// TwinCAT 3 PLC project Main
// ProgramVersion: 3.1.4024.0
// libraries:
//   mobject-core, * (mobject)
//   Tc2_Standard, * (Beckhoff Automation GmbH)
//   Tc2_System, * (Beckhoff Automation GmbH)
//   Tc2_Utilities, * (Beckhoff Automation GmbH)
//   Tc3_Module, * (Beckhoff Automation GmbH)
//   Tc3_Vision, * (Beckhoff Automation GmbH)
//   TcUnit, * (www.tcunit.org)
// project tree:
//   / PlcTask.TcTTO
//   POUs/Library/Animation/ I_Animation.TcIO, SpriteSheetAnimationFrames.TcPOU
//   POUs/Library/EL2574/DUT/ EL2574_Command.TcDUT
//   POUs/Library/EL2574/ EL2574_ExtendedMode.TcPOU, EL2574_CommandMode.TcPOU, I_EL2574_CommandMode.TcIO
//   POUs/Library/Functions/ HtmlColorCodeToRGBA.TcPOU
//   POUs/Library/Scene/ Scene.TcPOU
//   POUs/Library/ImageSerializer/Base/ ImageSerializer.TcPOU
//   POUs/Library/ImageSerializer/Interfaces/ I_ImageSerializer.TcIO
//   POUs/Library/ImageSerializer/Matrix/ MatrixImageSerializer.TcPOU
//   POUs/Library/ImageSerializer/Null/ NullImageSerializer.TcPOU
//   POUs/Library/PixelReader/ I_PixelReader.TcIO, EL2574PixelReader.TcPOU
//   POUs/ MAIN.TcPOU
//   Tests/ EL2574PixelReader_TestSuite.TcPOU, UnitTests.TcPOU
// real-time tasks:
//   TASK PlcTask: cycle T#700us, priority 20, ADS port 350
// I/O:
//   DEVICE Device 3 (EtherCAT), AmsNetId 172.18.232.102.4.1
//     Term 1 (EK1100) [EK1100 EtherCAT Coupler (2A E-Bus)]
//       Term 2 (EL2004) [EL2004 4Ch. Dig. Output 24V, 0.5A]
//       Term 3 (EL1014) [EL1014 4Ch. Dig. Input 24V, 10µs]
//       Term 4 (EL2574) [EL2574 4 Ch. Pixel LED Controller]
//         modules: SlotGroup 1 (Slot 1, 2) (1xASYNC), SlotGroup 1 (Slot 1, 2) (1xASYNC), SlotGroup 2 (Slot 3, 4) (1xASYNC), SlotGroup 2 (Slot 3, 4) (1xASYNC)
//       Term 5 (EL9011) [EL9011 End Terminal]
// variable links:
//   Main Instance <-> Device 3 (EtherCAT)/Term 1 (EK1100)/Term 3 (EL1014)
//     PlcTask Inputs/MAIN.switch <-> Channel 1/Input
//   Main Instance <-> Device 3 (EtherCAT)/Term 1 (EK1100)/Term 4 (EL2574)
//     PlcTask Inputs/MAIN.el2574_ch1.pdo.MDP5001_260_Input/MDP5001_260_Status <-> SlotGroup 1 (Slot 1, 2) (1xASYNC)/Status Channel 1/Status
//     PlcTask Inputs/MAIN.el2574_ch3.pdo.MDP5001_260_Input/MDP5001_260_Status <-> SlotGroup 2 (Slot 3, 4) (1xASYNC)/Status Channel 1/Status
//     PlcTask Outputs/MAIN.el2574_ch1.pdo.MDP5001_260_Output/MDP5001_260_Extended_Control <-> SlotGroup 1 (Slot 1, 2) (1xASYNC)/Extended Channel 1/Extended Control
//     PlcTask Outputs/MAIN.el2574_ch3.pdo.MDP5001_260_Output/MDP5001_260_Control <-> SlotGroup 2 (Slot 3, 4) (1xASYNC)/Control Channel 1/Control

CONFIGURATION Main
    RESOURCE PLC ON TwinCAT3
        TASK PlcTask(INTERVAL := T#700us, PRIORITY := 20);
        PROGRAM MAIN WITH PlcTask : MAIN;
    END_RESOURCE
END_CONFIGURATION

// ---- POUs/Library/EL2574/DUT/EL2574_Command.TcDUT
TYPE EL2574_Command :
STRUCT
	Send : BOOL;
	Update : BOOL;
	Command : USINT;
	Index : UINT;
	Length : UINT;
	Parameter : UINT;
	ColorRed : USINT;
	ColorGreen : USINT;
	ColorBlue : USINT;
	ColorWhite : USINT;
END_STRUCT
END_TYPE

// ---- POUs/Library/Animation/I_Animation.TcIO
INTERFACE I_Animation

PROPERTY PUBLIC CurrentFrameImage : ITcVnImage
GET
END_GET
END_PROPERTY

PROPERTY PUBLIC CurrentFrameIndex : UDINT
GET
END_GET
END_PROPERTY

PROPERTY PUBLIC IsAtLastFrame : BOOL
GET
END_GET
END_PROPERTY

METHOD PUBLIC MoveToStart
VAR_INPUT
END_VAR
END_METHOD

PROPERTY PUBLIC TotalFrameCount : UDINT
GET
END_GET
END_PROPERTY

METHOD PUBLIC TryMoveNext : BOOL
VAR_INPUT
END_VAR
END_METHOD

METHOD PUBLIC TryMovePrevious : BOOL
VAR_INPUT
END_VAR
END_METHOD

END_INTERFACE

// ---- POUs/Library/EL2574/I_EL2574_CommandMode.TcIO
INTERFACE I_EL2574_CommandMode

METHOD PUBLIC ClearAll : I_EL2574_CommandMode
VAR_INPUT
END_VAR
END_METHOD

METHOD PUBLIC ColorGradient2Point : I_EL2574_CommandMode
VAR_INPUT
	StartPosition : UINT;
	NumberOfPixels : UINT;
	Color1 : STRING(9);
	Color2 : STRING(9);
END_VAR
END_METHOD

METHOD PUBLIC ColorGradient3Point : I_EL2574_CommandMode
VAR_INPUT
	StartPosition : UINT;
	NumberOfPixels : UINT;
	Color1 : STRING(9);
	Color2 : STRING(9);
	Color3 : STRING(9);
END_VAR
END_METHOD

METHOD PUBLIC ColorGradient4Point : I_EL2574_CommandMode
VAR_INPUT
	StartPosition : UINT;
	NumberOfPixels : UINT;
	Color1 : STRING(9);
	Color2 : STRING(9);
	Color3 : STRING(9);
	Color4 : STRING(9);
END_VAR
END_METHOD

METHOD PUBLIC CopyPixels : I_EL2574_CommandMode
VAR_INPUT
	StartPosition : UINT;
	NumberOfPixels : UINT;
	TargetPosition : UINT;
END_VAR
END_METHOD

METHOD PUBLIC FillColor : I_EL2574_CommandMode
VAR_INPUT
	StartPosition : UINT;
	NumberOfPixels : UINT;
	Red : USINT;
	Green : USINT;
	Blue : USINT;
	White : USINT;
END_VAR
END_METHOD

METHOD PUBLIC Invert : I_EL2574_CommandMode
VAR_INPUT
	StartPosition : UINT;
	NumberOfPixels : UINT;
END_VAR
END_METHOD

METHOD PUBLIC MovePixels : I_EL2574_CommandMode
VAR_INPUT
	StartPosition : UINT;
	NumberOfPixels : UINT;
	TargetPosition : UINT;
END_VAR
END_METHOD

METHOD PUBLIC RotateLeft : I_EL2574_CommandMode
VAR_INPUT
	StartPosition : UINT;
	NumberOfPixels : UINT;
	Shift : UINT;
END_VAR
END_METHOD

METHOD PUBLIC RotateRight : I_EL2574_CommandMode
VAR_INPUT
	StartPosition : UINT;
	NumberOfPixels : UINT;
	Shift : UINT;
END_VAR
END_METHOD

METHOD PUBLIC Send : I_EL2574_CommandMode
VAR_INPUT
END_VAR
END_METHOD

METHOD PUBLIC SendAndUpdate : I_EL2574_CommandMode
VAR_INPUT
END_VAR
END_METHOD

METHOD PUBLIC Update : I_EL2574_CommandMode
VAR_INPUT
END_VAR
END_METHOD

END_INTERFACE

// ---- POUs/Library/ImageSerializer/Interfaces/I_ImageSerializer.TcIO
INTERFACE I_ImageSerializer

METHOD PUBLIC ConnectTo
VAR_INPUT
	ImageSerializer : I_ImageSerializer;
END_VAR
END_METHOD

METHOD PUBLIC GetTotalSerializablePixelCount : UDINT
VAR_INPUT
END_VAR
END_METHOD

PROPERTY PUBLIC PixelCount : UDINT
GET
END_GET
END_PROPERTY

METHOD PUBLIC TryGetPixel : BOOL
VAR_INPUT
	PixelIndex : UDINT;
	Reader : I_PixelReader;
END_VAR
END_METHOD

METHOD PUBLIC UpdateImage
VAR_INPUT
	Source : ITcVnImage;
END_VAR
END_METHOD

END_INTERFACE

// ---- POUs/Library/PixelReader/I_PixelReader.TcIO
INTERFACE I_PixelReader

PROPERTY PUBLIC Value : Reference to TcVnVector4_LREAL
GET
END_GET
END_PROPERTY

END_INTERFACE

// ---- POUs/MAIN.TcPOU
PROGRAM MAIN
VAR
	// demo triggers
	startAnimation : BOOL := TRUE;
	clear : BOOL := FALSE;
	mode : (RANDOM, NAUGHTY, NICE, SPECIAL) := RANDOM; // defaults each time to random
	
	// animations
	fireAnimation : SpriteSheetAnimationFrames(
		SpriteSheetFilePath := 'C:\temp\FireplaceAndFire_2_3_6.png',
		SpriteWidth := 32,
		SpriteHeight := 32,
		TotalSprites := 6,
		Columns := 2,
		Rows := 3
	);
	
	idleAnimation : SpriteSheetAnimationFrames(
		SpriteSheetFilePath := 'C:\temp\NaughtyOrNiceOutline_5_6_29.png',
		SpriteWidth := 32,
		SpriteHeight := 32,
		TotalSprites := 29,
		Columns := 5,
		Rows := 6
	);
	
	checkingList : SpriteSheetAnimationFrames(
		SpriteSheetFilePath := 'C:\temp\CheckingElfTree_4_4_16.png',
		SpriteWidth := 32,
		SpriteHeight := 32,
		TotalSprites := 16,
		Columns := 4,
		Rows := 4
	);
	
	anyCoverAnimation : SpriteSheetAnimationFrames(
		SpriteSheetFilePath := 'C:\temp\AnyCover_4_4_16.png',
		SpriteWidth := 32,
		SpriteHeight := 32,
		TotalSprites := 16,
		Columns := 4,
		Rows := 4
	);
	
	grinchAnimation : SpriteSheetAnimationFrames(
		SpriteSheetFilePath := 'C:\temp\Grinch_4_4_15.png',
		SpriteWidth := 32,
		SpriteHeight := 32,
		TotalSprites := 15,
		Columns := 4,
		Rows := 4
	);
	
	nicePresentAnimation : SpriteSheetAnimationFrames(
		SpriteSheetFilePath := 'C:\temp\NicePresent_4_5_19.png',
		SpriteWidth := 32,
		SpriteHeight := 32,
		TotalSprites := 19,
		Columns := 4,
		Rows := 5
	);
	
	specialAnimation : SpriteSheetAnimationFrames(
		SpriteSheetFilePath := 'C:\temp\sp_3_4_12.png',
		SpriteWidth := 32,
		SpriteHeight := 32,
		TotalSprites := 12,
		Columns := 3,
		Rows := 4
	);

	// matrix panels
	matrix1 : MatrixImageSerializer(Height := 16, Width := 16, X := 16, Y := 16, FlipX := FALSE, FlipY := TRUE, Rotate := TRUE);
	matrix2 : MatrixImageSerializer(Height := 16, Width := 16, X := 16, Y := 0, FlipX := FALSE, FlipY := TRUE, Rotate := TRUE); 
	matrix3 : MatrixImageSerializer(Height := 16, Width := 16, X := 0, Y := 0, FlipX := FALSE, FlipY := TRUE, Rotate := TRUE); 
	matrix4 : MatrixImageSerializer(Height := 16, Width := 16, X := 0, Y := 16, FlipX := FALSE, FlipY := TRUE, Rotate := TRUE); 
	
	// helpers
	scene : Scene;
	
	// hardware
	switch AT %I* : BOOL;
	el2574_ch1 : EL2574_ExtendedMode(TotalPixels := 1024); // you need to pass in the total number of pixels connected to the EK2574
	el2574_ch3 : EL2574_CommandMode(TotalPixels := 1024);
	
	// program variables
	initialized : BOOL;
	
	animationState : (
		IDLE_FWD, 
		IDLE_FWD_WAIT, 
		IDLE_BACKWARD, 
		IDLE_BACKWARD_WAIT, 
		CHECK_LIST, 
		COVER, 
		REVEAL_DECIDE, 
		REVEAL, 
		ACTUAL, 
		END_DELAY, 
		RESET
	) := RESET;
	
	actualAnimation : I_Animation;
	decision : USINT;
	
	ledState : (OFF, 
		OFF_WAIT, 
		IDLE_START, 
		IDLE_SEND_NEXT, 
		IDLE_WAIT, 
		CHECKING_START, 
		CHECKING_SEND_NEXT, 
		CHECKING_WAIT, 
		COVER_START,
		COVER_SEND_NEXT, 
		COVER_WAIT,
		REVEAL_NAUGHTY_START, 
		REVEAL_NAUGHTY_SEND_NEXT, 
		REVEAL_NAUGHTY_WAIT,
		REVEAL_NICE_START, 
		REVEAL_NICE_SEND_NEXT, 
		REVEAL_NICE_WAIT,
		REVEAL_SPECIAL_START, 
		REVEAL_SPECIAL_SEND_NEXT, 
		REVEAL_SPECIAL_WAIT
	) := OFF;
	
	animationRTrigger : R_TRIG;
	switchRTrigger : R_TRIG;
	triggerLedOff : R_TRIG;
	triggerLedIdle : R_TRIG;
	triggerLedChecking : R_TRIG;
	triggerLedCover : R_TRIG;
	triggerLedReveal : R_TRIG;
	
	// randomizer
	randomizer : USINT := 1; // very basic randomizer
	
	// counters 
	checklistCounter : INT; // this is just a simple setup to slow the animation down
	
	// timers
	idleForwardTimer : TON := (PT:=T#1S);
	idleBackwardTimer : TON := (PT:=T#2S);
	revealDecideTimer : TON := (PT:=T#1S);
	endDelayTimer : TON := (PT:=T#3S);
	fastLedTickerTimer : TON := (PT:=T#50MS);
	slowLedTickerTimer : TON := (PT:=T#200MS);
	
	// colors - variables so I can set them for testing. 	
	IDLE_COLOR_1 : STRING(9) := '04eeff';
	IDLE_COLOR_2 : STRING(9) := 'a206b1';
	IDLE_COLOR_3 : STRING(9) := '04eeff';
	
	CHECKING_COLOR_1 : STRING(9) := '0314f8';
	CHECKING_COLOR_2 : STRING(9) := '50aaa3';
	CHECKING_COLOR_3 : STRING(9) := '0314f8';

	COVER_COLOR_1 : STRING(9) := '09860f';
	COVER_COLOR_2 : STRING(9) := 'FF0000';
	COVER_COLOR_3 : STRING(9) := '09860f';
	
	REVEAL_NAUGHTY_COLOR_1 : STRING(9) := '09860f';
	REVEAL_NAUGHTY_COLOR_2 : STRING(9) := '000000';
	REVEAL_NAUGHTY_COLOR_3 : STRING(9) := '09860f';
	
	REVEAL_NICE_COLOR_1 : STRING(9) := 'FF0000';
	REVEAL_NICE_COLOR_2 : STRING(9) := '222222';
	REVEAL_NICE_COLOR_3 : STRING(9) := 'FF0000';
	
	REVEAL_SPECIAL_COLOR_1 : STRING(9) := 'f3ef16';
	REVEAL_SPECIAL_COLOR_2 : STRING(9) := 'FF0000';
	REVEAL_SPECIAL_COLOR_3 : STRING(9) := 'f3ef16';

END_VAR
VAR CONSTANT
	LED_STRIP_START : UINT := 120;
	LED_STRIP_LENGTH : UINT := 178;
END_VAR

(*

  _____ __  __ _____   ____  _____ _______       _   _ _______ _ 
 |_   _|  \/  |  __ \ / __ \|  __ \__   __|/\   | \ | |__   __| |
   | | | \  / | |__) | |  | | |__) | | |  /  \  |  \| |  | |  | |
   | | | |\/| |  ___/| |  | |  _  /  | | / /\ \ | . ` |  | |  | |
  _| |_| |  | | |    | |__| | | \ \  | |/ ____ \| |\  |  | |  |_|
 |_____|_|  |_|_|     \____/|_|  \_\ |_/_/    \_\_| \_|  |_|  (_)
 
Competition Clause: 

During the Beckhoff Christmas coding competition involving the EL2574 
LED controller terminal, if any Beckhoff subsidiaries use, borrow from, or are inspired
by this code for their own competition entry, they must acknowledge the inspiration by 
including the hashtag #codingbytes in any LinkedIn posts related to their competition entry. 
This requirement is in effect until the conclusion OF the competition on 25th December 2024.

*)

IF NOT initialized THEN
	// First setup the wiring of the units.  This must be in the order they are physically connected.
	matrix1.ConnectTo(matrix2);
	matrix2.ConnectTo(matrix3);
	matrix3.ConnectTo(matrix4);
	// that's initializing done!
	initialized := TRUE;
END_IF

// we wait here until the animation source image is loaded.
// i.e. we return, which prevents the program from progressing past this line.
IF NOT specialAnimation.TryLoad() OR NOT fireAnimation.TryLoad() OR NOT idleAnimation.TryLoad() OR NOT checkingList.TryLoad() OR NOT anyCoverAnimation.TryLoad() OR NOT grinchAnimation.TryLoad() OR NOT nicePresentAnimation.TryLoad() THEN
    RETURN;
END_IF

// basic clear trigger.  Set clear TRUE to clear the display
IF clear AND_THEN el2574_ch1.TrySendClearAll() THEN
	clear := FALSE;
END_IF

// if the startAnimation flag is triggered then force the state machine to RESET
animationRTrigger(Clk:=startAnimation);
IF animationRTrigger.Q THEN
	animationState := RESET;
END_IF

// if the "check" switch is pulled then move to CHECK_LIST if the program is running in idle
switchRTrigger(clk:=switch);
IF startAnimation AND switchRTrigger.Q AND (animationState = IDLE_FWD OR animationState = IDLE_FWD_WAIT OR animationState = IDLE_BACKWARD OR animationState = IDLE_BACKWARD_WAIT) THEN
	animationState := CHECK_LIST;
	decision := randomizer;
END_IF 

// animation state machine.
// this controls all of the image, animation and timinigs. 
IF startAnimation  AND NOT el2574_ch1.IsBusy THEN 
	
	CASE animationState OF
	
		IDLE_FWD :
			
			scene.Initalize(fireAnimation.CurrentFrameImage);
			scene.AddLayer(idleAnimation.CurrentFrameImage);
			
			IF NOT fireAnimation.TryMoveNext() THEN
				fireAnimation.MoveToStart();
			END_IF
			
			IF NOT idleAnimation.TryMoveNext() THEN
				animationState := IDLE_FWD_WAIT;
			END_IF
			
		IDLE_FWD_WAIT : 
		
			scene.Initalize(fireAnimation.CurrentFrameImage);
			scene.AddLayer(idleAnimation.CurrentFrameImage);
			
			IF NOT fireAnimation.TryMoveNext() THEN
				fireAnimation.MoveToStart();
			END_IF
		
			IF idleForwardTimer.Q THEN
				animationState := IDLE_BACKWARD;
			END_IF

		IDLE_BACKWARD :  
		
			scene.Initalize(fireAnimation.CurrentFrameImage);
			scene.AddLayer(idleAnimation.CurrentFrameImage);
			
			IF NOT fireAnimation.TryMoveNext() THEN
				fireAnimation.MoveToStart();
			END_IF
			
			IF NOT idleAnimation.TryMovePrevious() THEN
				animationState := IDLE_BACKWARD_WAIT;
			END_IF	

		IDLE_BACKWARD_WAIT : //	
		
			scene.Initalize(fireAnimation.CurrentFrameImage);
			scene.AddLayer(idleAnimation.CurrentFrameImage);
			
			IF NOT fireAnimation.TryMoveNext() THEN
				fireAnimation.MoveToStart();
			END_IF
		
			IF idleBackwardTimer.Q THEN
				animationState := IDLE_FWD;
			END_IF
			
		CHECK_LIST : 
		
			scene.Initalize(checkingList.CurrentFrameImage);
			
			IF checklistCounter > 2 AND_THEN NOT checkingList.TryMoveNext() THEN
				animationState := COVER;
			END_IF
			
			IF checklistCounter > 2 THEN
				checklistCounter := 0;
			ELSE 
				checklistCounter := checklistCounter + 1;
			END_IF
		
		COVER : //
		
			scene.Initalize(checkingList.CurrentFrameImage);
			scene.AddLayer(anyCoverAnimation.CurrentFrameImage);
			
			IF not anyCoverAnimation.TryMoveNext() THEN
				animationState := REVEAL_DECIDE;
			END_IF
			
		REVEAL_DECIDE : //
		
			IF revealDecideTimer.Q THEN
				
				// change mode to one of the two randoms.
				IF mode = RANDOM THEN
					IF decision > 5 THEN
						mode := NAUGHTY;
					ELSE
						mode := NICE;
					END_IF
				END_IF
				
				IF mode = NAUGHTY THEN
					actualAnimation := grinchAnimation;
				ELSIF mode = NICE THEN
					actualAnimation := nicePresentAnimation;
				ELSIF mode = SPECIAL THEN
					actualAnimation := specialAnimation;
				END_IF

				animationState := REVEAL;

			END_IF
		
		REVEAL : //
		
			scene.Initalize(actualAnimation.CurrentFrameImage);
			scene.AddLayer(anyCoverAnimation.CurrentFrameImage);
			
			IF NOT anyCoverAnimation.TryMovePrevious() THEN
				animationState := ACTUAL;
			END_IF
		
		ACTUAL : // 
		
			scene.Initalize(actualAnimation.CurrentFrameImage);
			
			IF NOT actualAnimation.TryMoveNext() THEN
				animationState := END_DELAY;
			END_IF
			
		END_DELAY : //
		
			IF endDelayTimer.Q THEN
				animationState := RESET;
			END_IF
			
		RESET : //
		
			idleAnimation.MoveToStart();
			checkingList.MoveToStart();
			anyCoverAnimation.MoveToStart();
			grinchAnimation.MoveToStart();
			nicePresentAnimation.MoveToStart();
			animationState := IDLE_FWD;
			mode := RANDOM;
	
	END_CASE
	
	matrix1.UpdateImage(scene.Image);
	el2574_ch1.TrySendPixelsFromSerializer(matrix1);
	
END_IF

// naughty, nice randomizer
randomizer := randomizer + 1;
IF randomizer > 10 THEN 
	randomizer := 1;
END_IF

// timers
idleForwardTimer(IN:=animationState=IDLE_FWD_WAIT);
idleBackwardTimer(IN:=animationState=IDLE_BACKWARD_WAIT);
revealDecideTimer(IN:=animationState=REVEAL_DECIDE);
endDelayTimer(IN:=animationState=END_DELAY);
fastLedTickerTimer(IN:=NOT fastLedTickerTimer.Q);
slowLedTickerTimer(IN:=NOT slowLedTickerTimer.Q);

// led state triggers
triggerLedOff(CLK := animationState=RESET);
IF triggerLedOff.Q THEN
	ledState := OFF;
END_IF

triggerLedIdle(CLK := animationState=IDLE_FWD);
IF triggerLedIdle.Q THEN
	ledState := IDLE_START;
END_IF

triggerLedChecking(CLK := animationState=CHECK_LIST);
IF triggerLedChecking.Q THEN
	ledState := CHECKING_START;
END_IF

triggerLedCover(CLK := animationState=COVER);
IF triggerLedCover.Q THEN
	ledState := COVER_START;
END_IF

triggerLedReveal(CLK := animationState=ACTUAL);
IF triggerLedReveal.Q THEN
	IF mode = NAUGHTY THEN
		ledState := REVEAL_NAUGHTY_START;
	ELSIF mode = NICE THEN
		ledState := REVEAL_NICE_START;
	ELSIF mode = SPECIAL THEN
		ledState := REVEAL_SPECIAL_START;
	END_IF
END_IF


// led state machine
CASE ledState OF
	
	OFF : //
	
		el2574_ch3.ClearAll();
		el2574_ch3.SendAndUpdate();
		ledState := OFF_WAIT;
	
	OFF_WAIT : // 
	
	IDLE_START : //
	
		el2574_ch3.ClearAll();
		el2574_ch3.ColorGradient3Point(LED_STRIP_START, 180, IDLE_COLOR_1, IDLE_COLOR_2, IDLE_COLOR_3);
		el2574_ch3.SendAndUpdate();
		ledState := IDLE_SEND_NEXT;
	
	IDLE_SEND_NEXT : //
	
		el2574_ch3.RotateRight(LED_STRIP_START, 180, 1); 
		el2574_ch3.SendAndUpdate();
		ledState := IDLE_WAIT;
		
	IDLE_WAIT : //
	
		IF NOT el2574_ch3.IsBusy AND fastLedTickerTimer.Q THEN
			ledState := IDLE_SEND_NEXT;
		END_IF
		
	CHECKING_START : //
	
		el2574_ch3.ClearAll();
		el2574_ch3.ColorGradient3Point(LED_STRIP_START, 180, CHECKING_COLOR_1, CHECKING_COLOR_2, CHECKING_COLOR_3);
		ledState := CHECKING_SEND_NEXT;
	
	CHECKING_SEND_NEXT : //
	
		el2574_ch3.RotateRight(LED_STRIP_START, 180, 1); 
		el2574_ch3.SendAndUpdate();
		ledState := CHECKING_WAIT;
	
	CHECKING_WAIT : //
	
		IF NOT el2574_ch3.IsBusy THEN
			ledState := CHECKING_SEND_NEXT;
		END_IF
		
	COVER_START : //
	
		el2574_ch3.ClearAll();
		el2574_ch3.ColorGradient3Point(LED_STRIP_START, 180, COVER_COLOR_1, COVER_COLOR_2, COVER_COLOR_3);
		ledState := COVER_SEND_NEXT;
	
	COVER_SEND_NEXT : //
	
		el2574_ch3.RotateRight(LED_STRIP_START, 180, 1); 
		el2574_ch3.SendAndUpdate();
		ledState := COVER_WAIT;
	
	COVER_WAIT : //
	
		IF NOT el2574_ch3.IsBusy THEN
			ledState := COVER_SEND_NEXT;
		END_IF
		
	REVEAL_NAUGHTY_START : //
	
		el2574_ch3.ClearAll();
		el2574_ch3.ColorGradient3Point(LED_STRIP_START, 180, REVEAL_NAUGHTY_COLOR_1, REVEAL_NAUGHTY_COLOR_2, REVEAL_NAUGHTY_COLOR_3);
		ledState := REVEAL_NAUGHTY_SEND_NEXT;
	
	REVEAL_NAUGHTY_SEND_NEXT : //
	
		el2574_ch3.RotateRight(LED_STRIP_START, 180, 1); 
		el2574_ch3.SendAndUpdate();
		ledState := REVEAL_NAUGHTY_WAIT;
	
	REVEAL_NAUGHTY_WAIT : //
	
		IF NOT el2574_ch3.IsBusy THEN
			ledState := REVEAL_NAUGHTY_SEND_NEXT;
		END_IF
		
	REVEAL_NICE_START : //
	
		el2574_ch3.ClearAll();
		el2574_ch3.ColorGradient3Point(LED_STRIP_START, 180, REVEAL_NICE_COLOR_1, REVEAL_NICE_COLOR_2, REVEAL_NICE_COLOR_3);
		ledState := REVEAL_NICE_SEND_NEXT;
	
	REVEAL_NICE_SEND_NEXT : //
	
		el2574_ch3.RotateRight(LED_STRIP_START, 180, 1); 
		el2574_ch3.SendAndUpdate();
		ledState := REVEAL_NICE_WAIT;
	
	REVEAL_NICE_WAIT : //
	
		IF NOT el2574_ch3.IsBusy THEN
			ledState := REVEAL_NICE_SEND_NEXT;
		END_IF
		
	REVEAL_SPECIAL_START : //
	
		el2574_ch3.ClearAll();
		el2574_ch3.ColorGradient3Point(LED_STRIP_START, 180, REVEAL_SPECIAL_COLOR_1, REVEAL_SPECIAL_COLOR_2, REVEAL_SPECIAL_COLOR_3);
		ledState := REVEAL_SPECIAL_SEND_NEXT;
	
	REVEAL_SPECIAL_SEND_NEXT : //
	
		el2574_ch3.RotateRight(LED_STRIP_START, 180, 1); 
		el2574_ch3.SendAndUpdate();
		ledState := REVEAL_SPECIAL_WAIT;
	
	REVEAL_SPECIAL_WAIT : //
	
		IF NOT el2574_ch3.IsBusy THEN
			ledState := REVEAL_SPECIAL_SEND_NEXT;
		END_IF
		
END_CASE

// cyclic call the terminal so that it can do it's job.
el2574_ch1.CyclicCall();
el2574_ch3.CyclicCall();

// unit tests
UnitTests();

END_PROGRAM

// ---- POUs/Library/Animation/SpriteSheetAnimationFrames.TcPOU
FUNCTION_BLOCK SpriteSheetAnimationFrames implements I_Animation
VAR
	spriteSheetFilePath : T_MAXSTRING;
	spriteWidth : UDINT;
	spriteHeight : UDINT;
	totalSprites : UDINT;
	columns : UDINT;
	rows : UDINT;
	spriteSheetImage : ITcVnImage;
	readImage: FB_VN_ReadImage;
	
	// animation variables
	_currentFrameIndex : UDINT;
	_currentFrameImage : ITcVnImage;
END_VAR

PROPERTY PUBLIC CurrentFrameImage : ITcVnImage
GET
CurrentFrameImage := _currentFrameImage;
END_GET
END_PROPERTY

PROPERTY PUBLIC CurrentFrameIndex : UDINT
GET
CurrentFrameIndex := _currentFrameIndex;
END_GET
END_PROPERTY

METHOD FB_init : BOOL
VAR_INPUT
	bInitRetains : BOOL; // if TRUE, the retain variables are initialized (warm start / cold start)
	bInCopyCode : BOOL;  // if TRUE, the instance afterwards gets moved into the copy code (online change)
	SpriteSheetFilePath : T_MAXSTRING;
	SpriteWidth : UDINT;
	SpriteHeight : UDINT;
	TotalSprites : UDINT;
	Columns : UDINT;
	Rows : UDINT;
END_VAR
THIS^.spriteSheetFilePath := SpriteSheetFilePath;
THIS^.spriteWidth := SpriteWidth;
THIS^.spriteHeight := SpriteHeight;
THIS^.totalSprites := TotalSprites;
THIS^.columns := Columns;
THIS^.rows := Rows;
END_METHOD

PROPERTY PUBLIC IsAtLastFrame : BOOL
GET
IF TotalFrameCount = 0 THEN
	IsAtLastFrame := TRUE;
	RETURN;
END_IF

IsAtLastFrame := CurrentFrameIndex = TotalFrameCount - 1;
END_GET
END_PROPERTY

METHOD PUBLIC MoveToStart
VAR_INPUT
END_VAR
_currentFrameIndex := 0;
TryGetSprite(_currentFrameIndex, _currentFrameImage);
END_METHOD

PROPERTY PUBLIC TotalFrameCount : UDINT
GET
TotalFrameCount := totalSprites;
END_GET
END_PROPERTY

METHOD PRIVATE TryGetSprite : BOOL
VAR_INPUT
	Index : UDINT;
	Destination : REFERENCE TO ITcVnImage;
END_VAR
VAR
	spriteX : UDINT;
	spriteY : UDINT;
	spriteColumn : UDINT;
	spriteRow : UDINT;
	result : HRESULT;
END_VAR
IF Index > TotalFrameCount - 1 THEN
	RETURN;
END_IF

spriteColumn := Index MOD columns;
spriteRow := Index / columns;

spriteX := spriteColumn * spriteWidth;
spriteY := spriteRow * spriteHeight;

result := F_VN_CopyImage(spriteSheetImage, _currentFrameImage, s_OK);
result := F_VN_SetRoi(spriteX, spriteY, spriteWidth, spriteHeight, _currentFrameImage, result);

TryGetSprite := Succeeded(result);
END_METHOD

METHOD PUBLIC TryLoad : BOOL
VAR
	i : UDINT;
END_VAR
// if we already have an image loaded, then we can early jump out as we know everything is done. 
IF spriteSheetImage <> 0 THEN
	TryLoad := TRUE;
	RETURN;
END_IF

IF spriteSheetFilePath = '' OR  spriteWidth = 0 OR spriteHeight = 0 OR totalSprites = 0 OR columns = 0 OR rows = 0 THEN
	// this is our sanity check, we return out if anything is bad.
	// if we pass this point we know we can use the variables confidently.
	RETURN;
END_IF

// we keep polling the read until an image is read.  If it faults due to error then we just sit here and never return true.
readImage(sFilePath := spriteSheetFilePath, ipDestImage := spriteSheetImage, bRead := TRUE, nTimeout := T#500MS);
IF readImage.bBusy THEN 
	RETURN;
END_IF

IF readImage.bError THEN 
	RETURN;
END_IF 

// at this point we should have an image, so we will do one final check before moving on.  
IF spriteSheetImage = 0 THEN
	RETURN;
END_IF

// we have made it this far, which means we need to set the CurrentFrameImage to the first part of the image and report as done. 
MoveToStart();
TryLoad := TRUE;
END_METHOD

METHOD PUBLIC TryMoveNext : BOOL
VAR_INPUT
END_VAR
IF _currentFrameIndex = TotalFrameCount - 1 THEN
	RETURN;
END_IF

_currentFrameIndex := _currentFrameIndex + 1;
TryMoveNext := TryGetSprite(_currentFrameIndex, _currentFrameImage);
END_METHOD

METHOD PUBLIC TryMovePrevious : BOOL
VAR_INPUT
END_VAR
IF _currentFrameIndex = 0 THEN
	RETURN;
END_IF

_currentFrameIndex := _currentFrameIndex - 1;
TryMovePrevious := TryGetSprite(_currentFrameIndex, _currentFrameImage);
END_METHOD

END_FUNCTION_BLOCK

// ---- POUs/Library/ImageSerializer/Matrix/MatrixImageSerializer.TcPOU
FUNCTION_BLOCK MatrixImageSerializer EXTENDS ImageSerializer
VAR
	height : UDINT;
	width : UDINT;
	x : UDINT;
	y : UDINT;
	flipRequired : BOOL;
	flipAxis : ETcVnFlipAxis;
	rotateRequired : BOOL;
	rotateAngle : ETcVnRotationAngle;
	
	image : ITcVnImage;
	live : ITcVnDisplayableImage; // used in this demo to show the image for the matrix
	_pixelCount : UDINT;
END_VAR

METHOD FB_init : BOOL
VAR_INPUT
	bInitRetains : BOOL; // if TRUE, the retain variables are initialized (warm start / cold start)
	bInCopyCode : BOOL;  // if TRUE, the instance afterwards gets moved into the copy code (online change)
	Height : UDINT;
	Width : UDINT;
	X : UDINT;
	Y : UDINT;
	FlipX : BOOL;
	FlipY : BOOL;
	Rotate : BOOL;
END_VAR
THIS^.height := Height;
THIS^.width := Width;
THIS^.x := X;
THIS^.y := Y;

IF FlipX AND FlipY THEN
	flipAxis := ETcVnFlipAxis.TCVN_FA_XY;
	flipRequired := TRUE;
ELSIF FlipX THEN
	flipAxis := ETcVnFlipAxis.TCVN_FA_X;
	flipRequired := TRUE;
ELSIF FlipY THEN
	flipAxis := ETcVnFlipAxis.TCVN_FA_Y;
	flipRequired := TRUE;
END_IF

IF Rotate THEN
	rotateRequired := TRUE;
	rotateAngle := ETcVnRotationAngle.TCVN_RA_90_DEG;
END_IF

Initialize();
END_METHOD

METHOD PRIVATE Initialize
VAR_INPUT
END_VAR
_pixelCount := width * height;
END_METHOD

METHOD PROTECTED OnTryGetPixel : BOOL
VAR_INPUT
	PixelIndex : UDINT;
	Reader : I_PixelReader;
END_VAR
VAR
	xPosition : UDINT;
	yPosition : UDINT;
END_VAR
IF width = 0 OR height = 0 THEN
	RETURN;
END_IF

xPosition := PixelIndex MOD width;
yPosition := PixelIndex / width;

// If it's an odd row, reverse the direction
IF yPosition MOD 2 = 1 THEN 
    xPosition := (width - 1) - xPosition;
END_IF

OnTryGetPixel := succeeded(F_VN_GetPixel(image, Reader.Value, xPosition, yPosition, s_OK));
END_METHOD

METHOD PROTECTED OnUpdateImage
VAR_INPUT
	Source : ITcVnImage;
END_VAR
VAR
	result : HRESULT;
END_VAR
result := F_VN_CopyImage(Source, image, s_OK);
result := F_VN_SetRoi(x, y, width, height, image, result);

IF flipRequired THEN
	result := F_VN_FlipImage(image, image, flipAxis, result);	
END_IF

IF rotateRequired THEN
	result := F_VN_RotateImage(image, image, rotateAngle, result);	
END_IF

IF Succeeded(result) THEN
	F_VN_CopyIntoDisplayableImage(image, live, s_ok);
	RETURN;
END_IF

// there was an error, so best to clear the internal image as it's no longer valid.
// but only if there was an image there in fht first place.

IF image = 0 THEN
	RETURN;
END_IF

image.TcRelease();
image := 0;
END_METHOD

{attribute 'monitoring' := 'call'}
PROPERTY PUBLIC PixelCount : UDINT
GET
PixelCount := _pixelCount;
END_GET
END_PROPERTY

END_FUNCTION_BLOCK

// ---- POUs/Library/ImageSerializer/Base/ImageSerializer.TcPOU
FUNCTION_BLOCK ABSTRACT ImageSerializer IMPLEMENTS I_ImageSerializer
VAR
	// using the null object pattern so that you no longer need to check to see if next is <> 0
	nullImageSerializer : NullImageSerializer;
	next : I_ImageSerializer := nullImageSerializer;
END_VAR

METHOD PUBLIC ConnectTo
VAR_INPUT
	ImageSerializer : I_ImageSerializer;
END_VAR
IF ImageSerializer = 0  THEN
	next := nullImageSerializer;
END_IF

IF ImageSerializer = next THEN
	RETURN;
END_IF

next := ImageSerializer;
END_METHOD

METHOD PUBLIC GetTotalSerializablePixelCount : UDINT
VAR_INPUT
END_VAR
GetTotalSerializablePixelCount := PixelCount + NextSerializer.GetTotalSerializablePixelCount();
END_METHOD

PROPERTY PUBLIC NextSerializer : I_ImageSerializer
GET
NextSerializer := next;
END_GET
END_PROPERTY

METHOD PROTECTED ABSTRACT OnTryGetPixel : BOOL
VAR_INPUT
	PixelIndex : UDINT;
	Reader : I_PixelReader;
END_VAR
END_METHOD

METHOD PROTECTED ABSTRACT OnUpdateImage
VAR_INPUT
	Source : ITcVnImage;
END_VAR
END_METHOD

PROPERTY PUBLIC ABSTRACT PixelCount : UDINT
GET
END_GET
END_PROPERTY

METHOD PUBLIC TryGetPixel : BOOL
VAR_INPUT
	PixelIndex : UDINT;
	Reader : I_PixelReader;
END_VAR
VAR
	newPixelIndex : UDINT;
END_VAR
IF PixelIndex > PixelCount - 1 THEN
	newPixelIndex := PixelIndex - PixelCount;
	TryGetPixel := NextSerializer.TryGetPixel(newPixelIndex, Reader);
	RETURN;
END_IF

TryGetPixel := OnTryGetPixel(PixelIndex, Reader);
END_METHOD

METHOD PUBLIC UpdateImage
VAR_INPUT
	Source : ITcVnImage;
END_VAR
IF Source = 0 THEN
	RETURN;
END_IF

OnUpdateImage(Source);
NextSerializer.UpdateImage(Source);
END_METHOD

END_FUNCTION_BLOCK

// ---- POUs/Library/ImageSerializer/Null/NullImageSerializer.TcPOU
FUNCTION_BLOCK NullImageSerializer IMPLEMENTS I_ImageSerializer
VAR
END_VAR

METHOD PUBLIC ConnectTo
VAR_INPUT
	ImageSerializer : I_ImageSerializer;
END_VAR
END_METHOD

METHOD PUBLIC GetTotalSerializablePixelCount : UDINT
VAR_INPUT
END_VAR
GetTotalSerializablePixelCount := 0;
END_METHOD

PROPERTY PUBLIC PixelCount : UDINT
GET
PixelCount := 0;
END_GET
END_PROPERTY

METHOD PUBLIC TryGetPixel : BOOL
VAR_INPUT
	PixelIndex : UDINT;
	Reader : I_PixelReader;
END_VAR
TryGetPixel := FALSE;
END_METHOD

METHOD PUBLIC UpdateImage
VAR_INPUT
	Source : ITcVnImage;
END_VAR
END_METHOD

END_FUNCTION_BLOCK

// ---- POUs/Library/Scene/Scene.TcPOU
FUNCTION_BLOCK Scene
VAR
	sceneImage : ITcVnImage;
END_VAR

METHOD PUBLIC AddLayer
VAR_INPUT
	Source : ITcVnImage;
END_VAR
VAR
	sourceHeight, currentHeight : UDINT;
	sourceWidth, currentWidth : UDINT;
	x, y : UDINT;
	currentPixel : TcVnVector4_LREAL;
END_VAR
IF sceneImage = 0 THEN
	RETURN;
END_IF

IF Source = 0 THEN 
	RETURN;
END_IF

IF FAILED(Source.GetHeight(sourceHeight)) THEN
	RETURN;
END_IF;

IF FAILED(sceneImage.GetHeight(currentHeight)) THEN
	RETURN;
END_IF;

IF FAILED(Source.GetWidth(sourceWidth)) THEN
	RETURN;
END_IF;

IF FAILED(sceneImage.GetWidth(currentWidth)) THEN
	RETURN;
END_IF;

IF sourceHeight > currentHeight THEN
	RETURN;
END_IF

IF sourceWidth > currentWidth THEN
	RETURN;
END_IF

FOR y := 0 TO sourceHeight - 1 DO
	FOR x := 0 TO sourceWidth - 1 DO
		
		IF SUCCEEDED(F_VN_GetPixel(Source, currentPixel, x, y, s_OK)) THEN
			IF currentPixel[0] = 0 AND currentPixel[1] = 0 AND currentPixel[2] = 0 THEN
				CONTINUE;
			END_IF
			F_VN_SetPixel(sceneImage, currentPixel,x,y,s_OK);	
		END_IF
	
	END_FOR
END_FOR
END_METHOD

PROPERTY PUBLIC Image : ITcVnImage
GET
Image := sceneImage;
END_GET
END_PROPERTY

METHOD PUBLIC Initalize
VAR_INPUT
	Source : ITcVnImage;
END_VAR
F_VN_CopyImage(Source, sceneImage, s_OK);
END_METHOD

END_FUNCTION_BLOCK

// ---- POUs/Library/EL2574/EL2574_ExtendedMode.TcPOU
FUNCTION_BLOCK EL2574_ExtendedMode
VAR
	totalPixels : UDINT;
	pdo : MDP5001_260_80E6114C;
	sendBuffer : ARRAY [0..MAX_PIXELS - 1] OF UDINT;
	sendSegmentCount : USINT;
	currentSegment : USINT;
	state : (IDLE, INITIALIZING, SEND_SEGMENT, TRIGGER_FRAME_SEND, WAIT_FOR_FRAME_SEND_COMPLETE, ERROR);
END_VAR
VAR CONSTANT
	MAX_PIXELS : UDINT := 2048;
END_VAR

METHOD PRIVATE CreateSendBufferFromSerializer
VAR_INPUT
	ImageSerializer : I_ImageSerializer;
END_VAR
VAR
	currentPixel : UDINT := 0;
	pixelReader : EL2574PixelReader;
END_VAR
WHILE ImageSerializer.TryGetPixel(currentPixel, pixelReader) DO
	sendBuffer[currentPixel] := pixelReader.ReadAsUdint();
	currentPixel := currentPixel + 1;
END_WHILE
END_METHOD

METHOD PUBLIC CyclicCall
VAR_INPUT
END_VAR
VAR
	totalSegments : UDINT;
END_VAR
CASE state OF
	
	IDLE : RETURN;
	ERROR : RETURN;
	
	INITIALIZING :
	
		// initialize local variables
		currentSegment := 0;
		totalSegments := totalPixels / 8;
		sendSegmentCount := UDINT_TO_USINT(totalSegments);
	
		// reset the card to a known state
		pdo.MDP5001_260_Output.MDP5001_260_Extended_Control.Index := 0;
		pdo.MDP5001_260_Output.MDP5001_260_Extended_Control.Send := FALSE;
		pdo.MDP5001_260_Output.MDP5001_260_Extended_Control.Update := FALSE;
		pdo.MDP5001_260_Output.MDP5001_260_Extended_Control.Write := FALSE;
		pdo.MDP5001_260_Output.MDP5001_260_Extended_Control.Segment.Element_0 := 0;
		pdo.MDP5001_260_Output.MDP5001_260_Extended_Control.Segment.Element_1 := 0;
		pdo.MDP5001_260_Output.MDP5001_260_Extended_Control.Segment.Element_2 := 0;
		pdo.MDP5001_260_Output.MDP5001_260_Extended_Control.Segment.Element_3 := 0;
		pdo.MDP5001_260_Output.MDP5001_260_Extended_Control.Segment.Element_4 := 0;
		pdo.MDP5001_260_Output.MDP5001_260_Extended_Control.Segment.Element_5 := 0;
		pdo.MDP5001_260_Output.MDP5001_260_Extended_Control.Segment.Element_6 := 0;
		pdo.MDP5001_260_Output.MDP5001_260_Extended_Control.Segment.Element_7 := 0;
		
		// start sending....
		state := SEND_SEGMENT;

	SEND_SEGMENT :
		
		pdo.MDP5001_260_Output.MDP5001_260_Extended_Control.Index := currentSegment;
		pdo.MDP5001_260_Output.MDP5001_260_Extended_Control.Segment.Element_0 := sendBuffer[currentSegment * 8 + 0];
		pdo.MDP5001_260_Output.MDP5001_260_Extended_Control.Segment.Element_1 := sendBuffer[currentSegment * 8 + 1];
		pdo.MDP5001_260_Output.MDP5001_260_Extended_Control.Segment.Element_2 := sendBuffer[currentSegment * 8 + 2];
		pdo.MDP5001_260_Output.MDP5001_260_Extended_Control.Segment.Element_3 := sendBuffer[currentSegment * 8 + 3];
		pdo.MDP5001_260_Output.MDP5001_260_Extended_Control.Segment.Element_4 := sendBuffer[currentSegment * 8 + 4];
		pdo.MDP5001_260_Output.MDP5001_260_Extended_Control.Segment.Element_5 := sendBuffer[currentSegment * 8 + 5];
		pdo.MDP5001_260_Output.MDP5001_260_Extended_Control.Segment.Element_6 := sendBuffer[currentSegment * 8 + 6];
		pdo.MDP5001_260_Output.MDP5001_260_Extended_Control.Segment.Element_7 := sendBuffer[currentSegment * 8 + 7];
		pdo.MDP5001_260_Output.MDP5001_260_Extended_Control.Write := TRUE;
		pdo.MDP5001_260_Output.MDP5001_260_Extended_Control.Execute := NOT pdo.MDP5001_260_Output.MDP5001_260_Extended_Control.Execute;
		
		IF currentSegment = sendSegmentCount THEN
			state := TRIGGER_FRAME_SEND;
		ELSE
			currentSegment := currentSegment + 1;
		END_IF
		
	TRIGGER_FRAME_SEND : 
	
		pdo.MDP5001_260_Output.MDP5001_260_Extended_Control.Write := FALSE;
		pdo.MDP5001_260_Output.MDP5001_260_Extended_Control.Update := TRUE;
		pdo.MDP5001_260_Output.MDP5001_260_Extended_Control.Send := TRUE;
		pdo.MDP5001_260_Output.MDP5001_260_Extended_Control.Execute := NOT pdo.MDP5001_260_Output.MDP5001_260_Extended_Control.Execute;
		
		state := WAIT_FOR_FRAME_SEND_COMPLETE;
		
	WAIT_FOR_FRAME_SEND_COMPLETE:
	
		IF NOT pdo.MDP5001_260_Input.MDP5001_260_Status.Busy THEN
			pdo.MDP5001_260_Output.MDP5001_260_Extended_Control.Update := FALSE;
			pdo.MDP5001_260_Output.MDP5001_260_Extended_Control.Send := FALSE;
			state := IDLE;
		END_IF

		
END_CASE
END_METHOD

METHOD FB_init : BOOL
VAR_INPUT
	bInitRetains : BOOL; // if TRUE, the retain variables are initialized (warm start / cold start)
	bInCopyCode : BOOL;  // if TRUE, the instance afterwards gets moved into the copy code (online change)
	TotalPixels : UDINT;
END_VAR
This^.totalPixels := TotalPixels;
END_METHOD

PROPERTY PUBLIC HasError : BOOL
GET
HasError := state = Error;
END_GET
END_PROPERTY

PROPERTY PUBLIC IsBusy : BOOL
GET
IsBusy := not(state = IDLE or_else state = ERROR);
END_GET
END_PROPERTY

METHOD PRIVATE ResetSendBuffer
VAR_INPUT
END_VAR
memset(ADR(sendBuffer), 0,SIZEOF(sendBuffer));
END_METHOD

METHOD PUBLIC TrySendClearAll : BOOL
VAR_INPUT
END_VAR
IF IsBusy THEN 
	RETURN;
END_IF

state := INITIALIZING;

ResetSendBuffer();
TrySendClearAll := TRUE;
END_METHOD

METHOD PUBLIC TrySendPixelsFromSerializer : BOOL
VAR_INPUT
	ImageSerializer : I_ImageSerializer;
END_VAR
IF IsBusy THEN 
	RETURN;
END_IF

IF ImageSerializer.GetTotalSerializablePixelCount() > totalPixels THEN 
	RETURN;
END_IF

state := INITIALIZING;

ResetSendBuffer();
CreateSendBufferFromSerializer(ImageSerializer);
TrySendPixelsFromSerializer := TRUE;
END_METHOD

END_FUNCTION_BLOCK

// ---- POUs/Library/PixelReader/EL2574PixelReader.TcPOU
FUNCTION_BLOCK EL2574PixelReader IMPLEMENTS I_PixelReader
VAR
	pixelValue : TcVnVector4_LREAL;
END_VAR

METHOD PUBLIC ReadAsUdint : UDINT
VAR_INPUT
END_VAR
VAR
	pixel : ARRAY [0..3] OF BYTE;
	pixelAsUint : UDINT;
END_VAR
pixel[0] := LREAL_TO_BYTE(value[0]);
pixel[1] := LREAL_TO_BYTE(value[1]);
pixel[2] := LREAL_TO_BYTE(value[2]);
pixel[3] := LREAL_TO_BYTE(value[3]);

memcpy(ADR(pixelAsUint), ADR(pixel),SIZEOF(pixelAsUint));
ReadAsUdint := pixelAsUint;
END_METHOD

PROPERTY PUBLIC Value : Reference to TcVnVector4_LREAL
GET
Value ref= pixelValue;
END_GET
END_PROPERTY

END_FUNCTION_BLOCK

// ---- POUs/Library/EL2574/EL2574_CommandMode.TcPOU
FUNCTION_BLOCK EL2574_CommandMode IMPLEMENTS I_EL2574_CommandMode
VAR
	totalPixels : UDINT;
	pdo : MDP5001_260_8D3B7340;
	commands : Queue;
	errored : BOOL;
END_VAR
VAR CONSTANT
	MAX_PIXELS : UDINT := 2048;
	COMMAND_NOP : USINT := 16#00;
	COMMAND_FILL : USINT := 16#01;
	COMMAND_CLEAR : USINT := 16#02;
	COMMAND_COPY : USINT := 16#03;
	COMMAND_MOVE : USINT := 16#04;
	COMMAND_ROTATE_LEFT : USINT := 16#05;
	COMMAND_ROTATE_RIGHT : USINT := 16#06;
	COMMAND_REVERSE : USINT := 16#07;
	COMMAND_GRADIENT_START : USINT := 16#08;
	COMMAND_GRADIENT_END : USINT := 16#09;
END_VAR

METHOD PUBLIC ClearAll : I_EL2574_CommandMode
VAR_INPUT
END_VAR
VAR
	command : EL2574_Command;
END_VAR
command.Send := FALSE;
command.Update := FALSE;
command.Command := COMMAND_CLEAR;
command.Index := 0;
command.Length := 0;
command.Parameter := 0;
command.ColorRed := 0;
command.ColorGreen := 0;
command.ColorBlue := 0;
command.ColorWhite := 0;

commands.Enqueue(command);

ClearAll := THIS^;
END_METHOD

METHOD PUBLIC ColorGradient2Point : I_EL2574_CommandMode
VAR_INPUT
	StartPosition : UINT;
	NumberOfPixels : UINT;
	Color1 : STRING(9);
	Color2 : STRING(9);
END_VAR
EnqueueGradientStart(StartPosition, NumberOfPixels, Color1);
EnqueueGradientEnd(StartPosition, NumberOfPixels, Color2);
ColorGradient2Point := THIS^;
END_METHOD

METHOD PUBLIC ColorGradient3Point : I_EL2574_CommandMode
VAR_INPUT
	StartPosition : UINT;
	NumberOfPixels : UINT;
	Color1 : STRING(9);
	Color2 : STRING(9);
	Color3 : STRING(9);
END_VAR
VAR
	segmentSize : UINT;
	finalSegmentSize : UINT;
	midpointStart : UINT;
END_VAR
IF NumberOfPixels < 3 THEN
	RETURN;
END_IF

segmentSize := NumberOfPixels / 2;
finalSegmentSize := NumberOfPixels - segmentSize;
midpointStart := StartPosition + segmentSize;

EnqueueGradientStart(StartPosition, segmentSize, Color1);
EnqueueGradientEnd(StartPosition, segmentSize, Color2);
EnqueueGradientStart(midpointStart, finalSegmentSize, Color2);
EnqueueGradientEnd(midpointStart, finalSegmentSize, Color3);

ColorGradient3Point := THIS^;
END_METHOD

METHOD PUBLIC ColorGradient4Point : I_EL2574_CommandMode
VAR_INPUT
	StartPosition : UINT;
	NumberOfPixels : UINT;
	Color1 : STRING(9);
	Color2 : STRING(9);
	Color3 : STRING(9);
	Color4 : STRING(9);
END_VAR
VAR
	segmentSize : UINT;
	finalSegmentSize : UINT;
	firstThirdStart : UINT;
	secondThirdStart : UINT;
END_VAR
IF NumberOfPixels < 3 THEN
	RETURN;
END_IF

segmentSize := NumberOfPixels / 3;

firstThirdStart := StartPosition + segmentSize;
secondThirdStart := StartPosition + segmentSize * 2;

finalSegmentSize := NumberOfPixels - (segmentSize * 2);

EnqueueGradientStart(StartPosition, segmentSize, Color1);
EnqueueGradientEnd(StartPosition, segmentSize, Color2);
EnqueueGradientStart(firstThirdStart, segmentSize, Color2);
EnqueueGradientEnd(firstThirdStart, segmentSize, Color3);
EnqueueGradientStart(secondThirdStart, finalSegmentSize, Color3);
EnqueueGradientEnd(secondThirdStart, finalSegmentSize, Color4);

ColorGradient4Point := THIS^;
END_METHOD

METHOD PUBLIC CopyPixels : I_EL2574_CommandMode
VAR_INPUT
	StartPosition : UINT;
	NumberOfPixels : UINT;
	TargetPosition : UINT;
END_VAR
VAR
	command : EL2574_Command;
END_VAR
command.Send := FALSE;
command.Update := FALSE;
command.Command := COMMAND_COPY;
command.Index := StartPosition;
command.Length := NumberOfPixels;
command.Parameter := TargetPosition;
command.ColorRed := 0;
command.ColorGreen := 0;
command.ColorBlue := 0;
command.ColorWhite := 0;

commands.Enqueue(command);

CopyPixels := THIS^;
END_METHOD

METHOD PUBLIC CyclicCall
VAR_INPUT
END_VAR
VAR
	sendCommand : EL2574_Command;
END_VAR
IF pdo.MDP5001_260_Input.MDP5001_260_Status.Busy THEN
	RETURN;
END_IF

IF pdo.MDP5001_260_Input.MDP5001_260_Status.Transmit THEN
	RETURN;
END_IF

IF commands.IsEmpty THEN 
	RETURN;
END_IF

IF NOT commands.TryDequeue(sendCommand) THEN
	errored := TRUE;
	RETURN;
END_IF

pdo.MDP5001_260_Output.MDP5001_260_Control.Send := sendCommand.Send;
pdo.MDP5001_260_Output.MDP5001_260_Control.Update := sendCommand.Update;
pdo.MDP5001_260_Output.MDP5001_260_Control.Command := sendCommand.Command;
pdo.MDP5001_260_Output.MDP5001_260_Control.Index := sendCommand.Index;
pdo.MDP5001_260_Output.MDP5001_260_Control.Length := sendCommand.Length;
pdo.MDP5001_260_Output.MDP5001_260_Control.Parameter := sendCommand.Parameter;
pdo.MDP5001_260_Output.MDP5001_260_Control.Color.Red := sendCommand.ColorRed;
pdo.MDP5001_260_Output.MDP5001_260_Control.Color.Green := sendCommand.ColorGreen;
pdo.MDP5001_260_Output.MDP5001_260_Control.Color.Blue := sendCommand.ColorBlue;
pdo.MDP5001_260_Output.MDP5001_260_Control.Color.White := sendCommand.ColorWhite;
pdo.MDP5001_260_Output.MDP5001_260_Control.Execute := NOT pdo.MDP5001_260_Output.MDP5001_260_Control.Execute;
END_METHOD

METHOD PRIVATE EnqueueGradientEnd
VAR_INPUT
	StartPosition : UINT;
	NumberOfPixels : UINT;
	Color : STRING(9);
END_VAR
VAR
	convertedColor : ARRAY [0..3] OF USINT;
	command : EL2574_Command;
END_VAR
convertedColor := HtmlColorCodeToRGBA(Color);

command.Send := FALSE;
command.Update := FALSE;
command.Command := COMMAND_GRADIENT_END;
command.Index := StartPosition;
command.Length := NumberOfPixels;
command.Parameter := 0;
command.ColorRed := convertedColor[0];
command.ColorGreen := convertedColor[1];
command.ColorBlue := convertedColor[2];
command.ColorWhite := convertedColor[3];

commands.Enqueue(command);
END_METHOD

METHOD PRIVATE EnqueueGradientStart
VAR_INPUT
	StartPosition : UINT;
	NumberOfPixels : UINT;
	Color : STRING(9);
END_VAR
VAR
	convertedColor : ARRAY [0..3] OF USINT;
	command : EL2574_Command;
END_VAR
convertedColor := HtmlColorCodeToRGBA(Color);

command.Send := FALSE;
command.Update := FALSE;
command.Command := COMMAND_GRADIENT_START;
command.Index := StartPosition;
command.Length := NumberOfPixels;
command.Parameter := 0;
command.ColorRed := convertedColor[0];
command.ColorGreen := convertedColor[1];
command.ColorBlue := convertedColor[2];
command.ColorWhite := convertedColor[3];

commands.Enqueue(command);
END_METHOD

METHOD FB_init : BOOL
VAR_INPUT
	bInitRetains : BOOL; // if TRUE, the retain variables are initialized (warm start / cold start)
	bInCopyCode : BOOL;  // if TRUE, the instance afterwards gets moved into the copy code (online change)
	TotalPixels : UDINT;
END_VAR
This^.totalPixels := TotalPixels;
END_METHOD

METHOD PUBLIC FillColor : I_EL2574_CommandMode
VAR_INPUT
	StartPosition : UINT;
	NumberOfPixels : UINT;
	Red : USINT;
	Green : USINT;
	Blue : USINT;
	White : USINT;
END_VAR
VAR
	command : EL2574_Command;
END_VAR
command.Send := FALSE;
command.Update := FALSE;
command.Command := COMMAND_FILL;
command.Index := StartPosition;
command.Length := NumberOfPixels;
command.Parameter := 0;
command.ColorRed := Red;
command.ColorGreen := Green;
command.ColorBlue := Blue;
command.ColorWhite := White;

commands.Enqueue(command);

FillColor := THIS^;
END_METHOD

PROPERTY PUBLIC HasError : BOOL
GET
HasError := errored;
END_GET
END_PROPERTY

METHOD PUBLIC Invert : I_EL2574_CommandMode
VAR_INPUT
	StartPosition : UINT;
	NumberOfPixels : UINT;
END_VAR
VAR
	command : EL2574_Command;
END_VAR
command.Send := FALSE;
command.Update := FALSE;
command.Command := COMMAND_REVERSE;
command.Index := StartPosition;
command.Length := NumberOfPixels;
command.Parameter := 0;
command.ColorRed := 0;
command.ColorGreen := 0;
command.ColorBlue := 0;
command.ColorWhite := 0;

commands.Enqueue(command);

Invert := THIS^;
END_METHOD

PROPERTY PUBLIC IsBusy : BOOL
GET
IsBusy := pdo.MDP5001_260_Input.MDP5001_260_Status.Busy OR NOT commands.IsEmpty;
END_GET
END_PROPERTY

METHOD PUBLIC MovePixels : I_EL2574_CommandMode
VAR_INPUT
	StartPosition : UINT;
	NumberOfPixels : UINT;
	TargetPosition : UINT;
END_VAR
VAR
	command : EL2574_Command;
END_VAR
command.Send := FALSE;
command.Update := FALSE;
command.Command := COMMAND_MOVE;
command.Index := StartPosition;
command.Length := NumberOfPixels;
command.Parameter := TargetPosition;
command.ColorRed := 0;
command.ColorGreen := 0;
command.ColorBlue := 0;
command.ColorWhite := 0;

commands.Enqueue(command);

MovePixels := THIS^;
END_METHOD

METHOD PUBLIC RotateLeft : I_EL2574_CommandMode
VAR_INPUT
	StartPosition : UINT;
	NumberOfPixels : UINT;
	Shift : UINT;
END_VAR
VAR
	command : EL2574_Command;
END_VAR
command.Send := FALSE;
command.Update := FALSE;
command.Command := COMMAND_ROTATE_LEFT;
command.Index := StartPosition;
command.Length := NumberOfPixels;
command.Parameter := Shift;
command.ColorRed := 0;
command.ColorGreen := 0;
command.ColorBlue := 0;
command.ColorWhite := 0;

commands.Enqueue(command);

RotateLeft := THIS^;
END_METHOD

METHOD PUBLIC RotateRight : I_EL2574_CommandMode
VAR_INPUT
	StartPosition : UINT;
	NumberOfPixels : UINT;
	Shift : UINT;
END_VAR
VAR
	command : EL2574_Command;
END_VAR
command.Send := FALSE;
command.Update := FALSE;
command.Command := COMMAND_ROTATE_RIGHT;
command.Index := StartPosition;
command.Length := NumberOfPixels;
command.Parameter := Shift;
command.ColorRed := 0;
command.ColorGreen := 0;
command.ColorBlue := 0;
command.ColorWhite := 0;

commands.Enqueue(command);

RotateRight := THIS^;
END_METHOD

METHOD PUBLIC Send : I_EL2574_CommandMode
VAR_INPUT
END_VAR
VAR
	command : EL2574_Command;
END_VAR
command.Send := TRUE;
command.Update := FALSE;
command.Command := COMMAND_NOP;
command.Index := 0;
command.Length := 0;
command.Parameter := 0;
command.ColorRed := 0;
command.ColorGreen := 0;
command.ColorBlue := 0;
command.ColorWhite := 0;

commands.Enqueue(command);

Send := THIS^;
END_METHOD

METHOD PUBLIC SendAndUpdate : I_EL2574_CommandMode
VAR_INPUT
END_VAR
VAR
	command : EL2574_Command;
END_VAR
command.Send := TRUE;
command.Update := TRUE;
command.Command := COMMAND_NOP;
command.Index := 0;
command.Length := 0;
command.Parameter := 0;
command.ColorRed := 0;
command.ColorGreen := 0;
command.ColorBlue := 0;
command.ColorWhite := 0;

commands.Enqueue(command);

SendAndUpdate := THIS^;
END_METHOD

METHOD PUBLIC Update : I_EL2574_CommandMode
VAR_INPUT
END_VAR
VAR
	command : EL2574_Command;
END_VAR
command.Send := FALSE;
command.Update := TRUE;
command.Command := COMMAND_NOP;
command.Index := 0;
command.Length := 0;
command.Parameter := 0;
command.ColorRed := 0;
command.ColorGreen := 0;
command.ColorBlue := 0;
command.ColorWhite := 0;

commands.Enqueue(command);

Update := THIS^;
END_METHOD

END_FUNCTION_BLOCK

// ---- POUs/Library/Functions/HtmlColorCodeToRGBA.TcPOU
FUNCTION HtmlColorCodeToRGBA : ARRAY [0..3] OF USINT
VAR_INPUT
	ColorCode : STRING(9);
END_VAR
VAR
	toConvert : STRING;
	converted : ARRAY [0..3] OF USINT;
END_VAR

// allow the user to pass in the # as optional
IF FIND(ColorCode,'#') = 1 THEN
	toConvert := right(ColorCode, len(ColorCode)-1);
ELSE
	toConvert := ColorCode;
END_IF

// check for a valid string, i.e. must be 6 or 8 chars long.
IF NOT(len(toConvert) = 6 OR len(toConvert) = 8) THEN
	RETURN;
END_IF

// allow 6 or 8 hex codes
IF len(toConvert) = 6 THEN
	toConvert := concat(toConvert,'00');
END_IF

HEXSTR_TO_DATA( toConvert, ADR(converted), SIZEOF(converted));
HtmlColorCodeToRGBA := converted;

END_FUNCTION

// ---- Tests/UnitTests.TcPOU
PROGRAM UnitTests
VAR
	el2574PixelReader_TestSuite : EL2574PixelReader_TestSuite;
END_VAR

TcUnit.RUN();

END_PROGRAM

// ---- Tests/EL2574PixelReader_TestSuite.TcPOU
FUNCTION_BLOCK EL2574PixelReader_TestSuite EXTENDS TcUnit.FB_TestSuite

TestReadAsUdint_Blank();
TestReadAsUdint_Blue();
TestReadAsUdint_Green();
TestReadAsUdint_Red();

METHOD PUBLIC TestReadAsUdint_Blank
VAR
	pixelReader : EL2574PixelReader;
	pixel : TcVnVector4_LREAL := [0,0,0,0];
	actual : UDINT;
	expected : UDINT := 0; 
END_VAR
TEST('TestReadAsUdint_Blank');

pixelReader.Value := pixel;
actual := pixelReader.ReadAsUdint();

AssertEquals(
	Actual := actual,
	Expected := expected,
	Message := 'Did not return the correct pixel value'
);

TEST_FINISHED();
END_METHOD

METHOD PUBLIC TestReadAsUdint_Blue
VAR
	pixelReader : EL2574PixelReader;
	pixel : TcVnVector4_LREAL := [0,0,255,0];
	actual : UDINT;
	expected : UDINT := 16#00FF0000;
END_VAR
TEST('TestReadAsUdint_Blue');

pixelReader.Value := pixel;
actual := pixelReader.ReadAsUdint();

AssertEquals(
	Actual := actual,
	Expected := expected,
	Message := 'Did not return the correct pixel value'
);

TEST_FINISHED();
END_METHOD

METHOD PUBLIC TestReadAsUdint_Green
VAR
	pixelReader : EL2574PixelReader;
	pixel : TcVnVector4_LREAL := [0,255,0,0];
	actual : UDINT;
	expected : UDINT := 16#0000FF00;
END_VAR
TEST('TestReadAsUdint_Red');

pixelReader.Value := pixel;
actual := pixelReader.ReadAsUdint();

AssertEquals(
	Actual := actual,
	Expected := expected,
	Message := 'Did not return the correct pixel value'
);

TEST_FINISHED();
END_METHOD

METHOD PUBLIC TestReadAsUdint_Red
VAR
	pixelReader : EL2574PixelReader;
	pixel : TcVnVector4_LREAL := [255,0,0,0];
	actual : UDINT;
	expected : UDINT := 16#000000FF;
END_VAR
TEST('TestReadAsUdint_Red');

pixelReader.Value := pixel;
actual := pixelReader.ReadAsUdint();

AssertEquals(
	Actual := actual,
	Expected := expected,
	Message := 'Did not return the correct pixel value'
);

TEST_FINISHED();
END_METHOD

END_FUNCTION_BLOCK
